FUNCTION_BLOCK MUX_DATE_AND_TIME (* See MUX_ANY *)
  (* Standard: 61131-3 *)
  (* Version 0.0, 2004-12-15, JHC, Rockwell Automation, Converted from SRC format. *)
  (* Compiler header: package fb.rt.plc.select; *)
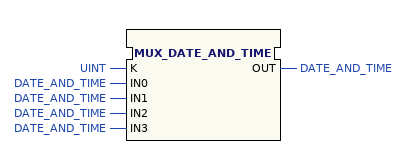
  VAR_INPUT
    K : UINT;
    IN0 : DATE_AND_TIME;
    IN1 : DATE_AND_TIME;
    IN2 : DATE_AND_TIME;
    IN3 : DATE_AND_TIME;
  END_VAR
  VAR_OUTPUT
    OUT : DATE_AND_TIME;
  END_VAR
END_FUNCTION_BLOCK
